(* CODESYS project Estampadora.project
   Title: RepasoEjercicio1
   Version: 0.0.0.0
   Author: bou

Project tree, tasks and I/O mapping:
  PLC_Cabecera_linea_ : TM241CE40R, Schneider Electric, order no. TM241CE40R, version 4.0.6.18
    application Application
      task MAST (cyclic, interval 30 ms, priority 15, watchdog 100 ms x 10) calls Control_Grafcet
      global variables GVL
      visualisation Interface_Main
      program Control_Grafcet [SFC]
      image pool ImagePool
      program Moves [LD]
      trace Registro de traza (task MAST): DIRMAQUINA
    DI : Digital Inputs, Schneider Electric, version 4.0.6.18
        input  idwDI_IDW0 : DWORD  // IDW0
        input  ibDI_IB1 : BYTE  // IB1
    DQ : Digital Outputs, Schneider Electric, version 4.0.6.18
        output qwDQ_QW0 : WORD  // QW0
        output qbDQ_QB1 : BYTE  // QB1
    Counters : Counters, Schneider Electric, version 4.0.6.18
    Pulse_Generators : Pulse Generators, Schneider Electric, version 4.0.6.18
    Cartridge_1 : Cartridge, Schneider Electric, version 4.0.6.18
    Cartridge_2 : Cartridge, Schneider Electric, version 4.0.6.18
    IO_Bus : IO bus - TM3, Schneider Electric, version 4.0.6.18
    COM_Bus : COM bus, Schneider Electric, version 4.0.6.18
    Ethernet_1 : Ethernet Network, Schneider Electric, version 4.0.6.18
        settings: IPAddress = [172, 16, 191, 108]; SubnetMask = [255, 255, 255, 0]; GatewayAddress = [172, 16, 191, 1]; WebServer = TRUE; FTP Server = TRUE; SoMachine Protocol = TRUE; Modbus Server = TRUE; NetManage Protocol = TRUE; SNMP protocol = TRUE; Enable Routing = FALSE; WebVisu protocol = TRUE; DHCP Server Active = FALSE
    Serial_Line_1 : Serial line, Schneider Electric, version 4.0.6.18
    Serial_Line_2 : Serial line, Schneider Electric, version 4.0.6.18
  text list GlobalTextList
*)

// PLC_Cabecera_linea_/Application/GVL
VAR_GLOBAL
END_VAR
VAR_GLOBAL
	PULSADOR AT %IX0.0: BOOL;
	S1_INI AT %IX0.1: BOOL;
	S2_FIN AT %IX0.2: BOOL;
	ARRIBA AT %IX0.3: BOOL;
	ABAJO AT %IX0.4: BOOL;
	INTERRUPTOR AT %IX0.5: BOOL;
	POWER AT %QX1.0: BOOL;
	CINTA_ABANCE AT %QX0.4: BOOL;
	CINTA_RETROCESO AT %QX0.5: BOOL;
	MAQUINA_ARRIBA AT %QX0.6: BOOL;
	MAQUINA_ABAJO AT %QX0.7: BOOL;
	ENCENDIDO: BOOL;
	INICIO: BOOL;
END_VAR

// PLC_Cabecera_linea_/Application/Control_Grafcet
PROGRAM Control_Grafcet
VAR
END_VAR

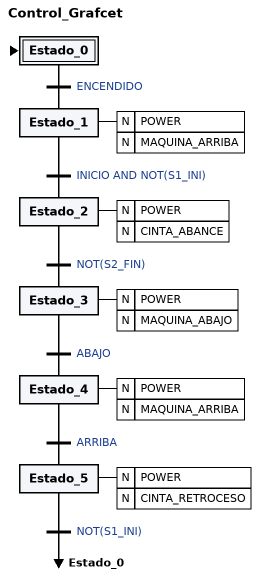
INITIAL_STEP Estado_0:
END_STEP
TRANSITION FROM Estado_0 TO Estado_1
    := ENCENDIDO;
END_TRANSITION
STEP Estado_1:
    POWER(N);
    MAQUINA_ARRIBA(N);
END_STEP
TRANSITION FROM Estado_1 TO Estado_2
    := INICIO AND NOT(S1_INI);
END_TRANSITION
STEP Estado_2:
    POWER(N);
    CINTA_ABANCE(N);
END_STEP
TRANSITION FROM Estado_2 TO Estado_3
    := NOT(S2_FIN);
END_TRANSITION
STEP Estado_3:
    POWER(N);
    MAQUINA_ABAJO(N);
END_STEP
TRANSITION FROM Estado_3 TO Estado_4
    := ABAJO;
END_TRANSITION
STEP Estado_4:
    POWER(N);
    MAQUINA_ARRIBA(N);
END_STEP
TRANSITION FROM Estado_4 TO Estado_5
    := ARRIBA;
END_TRANSITION
STEP Estado_5:
    POWER(N);
    CINTA_RETROCESO(N);
END_STEP
TRANSITION FROM Estado_5 TO Estado_0
    := NOT(S1_INI);
END_TRANSITION

END_PROGRAM

// PLC_Cabecera_linea_/Application/Moves
PROGRAM Moves
VAR
	Estampa: UINT;
	My_S1_INI: BOOL;
	My_S2_FIN: BOOL;
	
END_VAR
VAR // added by the converter: edge detectors and wires of the graphical bodies
    _w1, _w2, _w3 : BOOL;
END_VAR

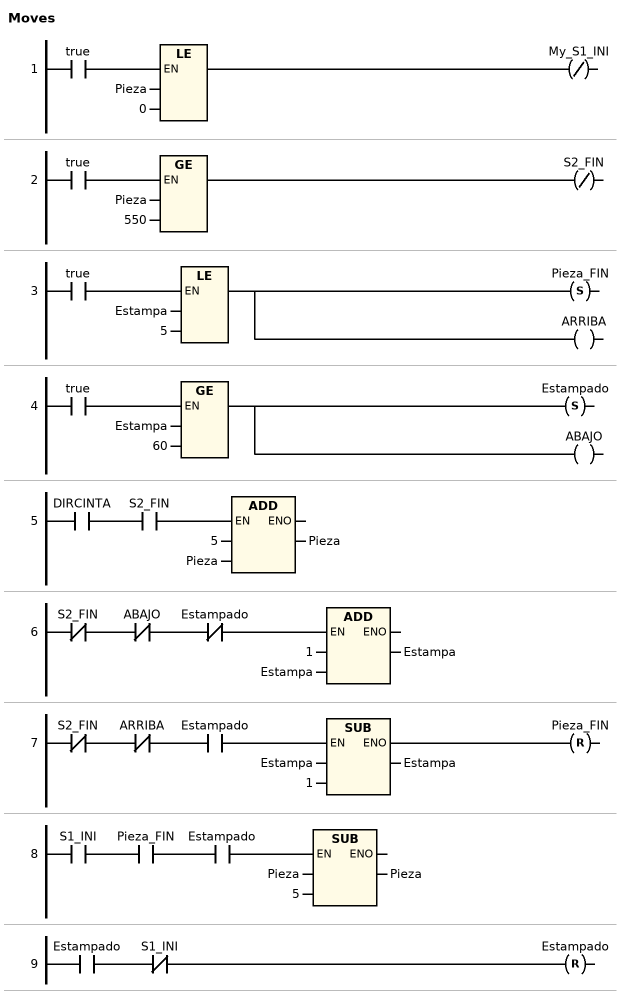
// NETWORK 1
My_S1_INI := NOT (true AND Pieza <= 0);

// NETWORK 2
S2_FIN := NOT (true AND Pieza >= 550);

// NETWORK 3
_w1 := true AND Estampa <= 5;
Pieza_FIN S= _w1;
ARRIBA := _w1;

// NETWORK 4
_w2 := true AND Estampa >= 60;
Estampado S= _w2;
ABAJO := _w2;

// NETWORK 5
IF DIRCINTA AND S2_FIN THEN Pieza := 5 + Pieza; END_IF

// NETWORK 6
IF NOT S2_FIN AND NOT ABAJO AND NOT Estampado THEN Estampa := 1 + Estampa; END_IF

// NETWORK 7
_w3 := NOT S2_FIN AND NOT ARRIBA AND Estampado;
IF _w3 THEN Estampa := Estampa - 1; END_IF
Pieza_FIN R= _w3;

// NETWORK 8
IF S1_INI AND Pieza_FIN AND Estampado THEN Pieza := Pieza - 5; END_IF

// NETWORK 9
Estampado R= Estampado AND NOT S1_INI;

END_PROGRAM

// PLC_Cabecera_linea_/Application/Interface_Main
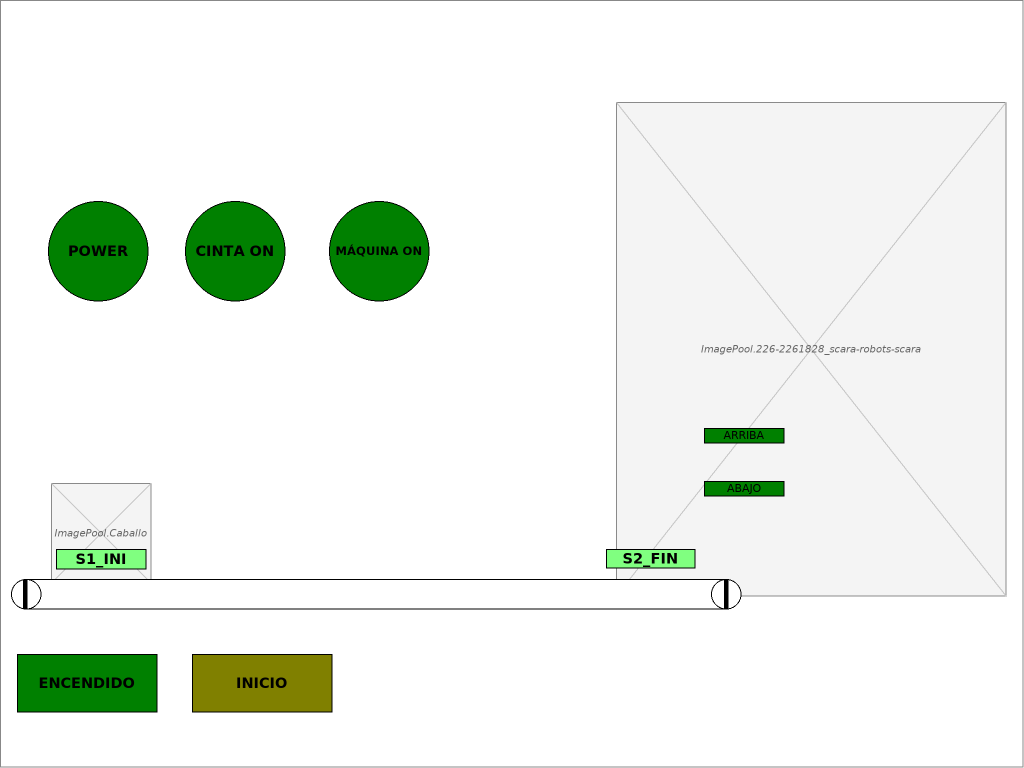
VISUALIZATION Interface_Main  // 1024x768
    Image (51,483 100x100), image: ImagePool.Caballo
        p3560616238: Pieza
    Rectangle (645,370 10x70)
        p2738717112: Estampa
    Image (616,102 390x494), image: ImagePool.226-2261828_scara-robots-scara
    Rectangle (17,654 140x58), "ENCENDIDO", colour toggle: Control_Grafcet.ENCENDIDO
        tap Control_Grafcet.ENCENDIDO
    Rectangle (192,654 140x58), "INICIO", colour toggle: Control_Grafcet.INICIO
        tap Control_Grafcet.INICIO
    Rectangle (26,579 700x30)
    Ellipse (711,579 30x30)
    Ellipse (11,579 30x30)
    Rectangle (56,549 90x20), "S1_INI", colour toggle: Control_Grafcet.S1_INI
    Rectangle (606,549 89x19), "S2_FIN", colour toggle: Control_Grafcet.S2_FIN
    Rectangle (704,428 80x15), "ARRIBA", colour toggle: ARRIBA
    Rectangle (704,481 80x15), "ABAJO", colour toggle: ABAJO
    Ellipse (48,201 100x100), "POWER", colour toggle: POWER
    Ellipse (185,201 100x100), "CINTA ON"
    Ellipse (329,201 100x100), "MÁQUINA ON"
    Rectangle (724,580 4x28)
        p2858320360: Pieza
    Rectangle (23,580 4x28)
        p2858320360: Pieza
END_VISUALIZATION
